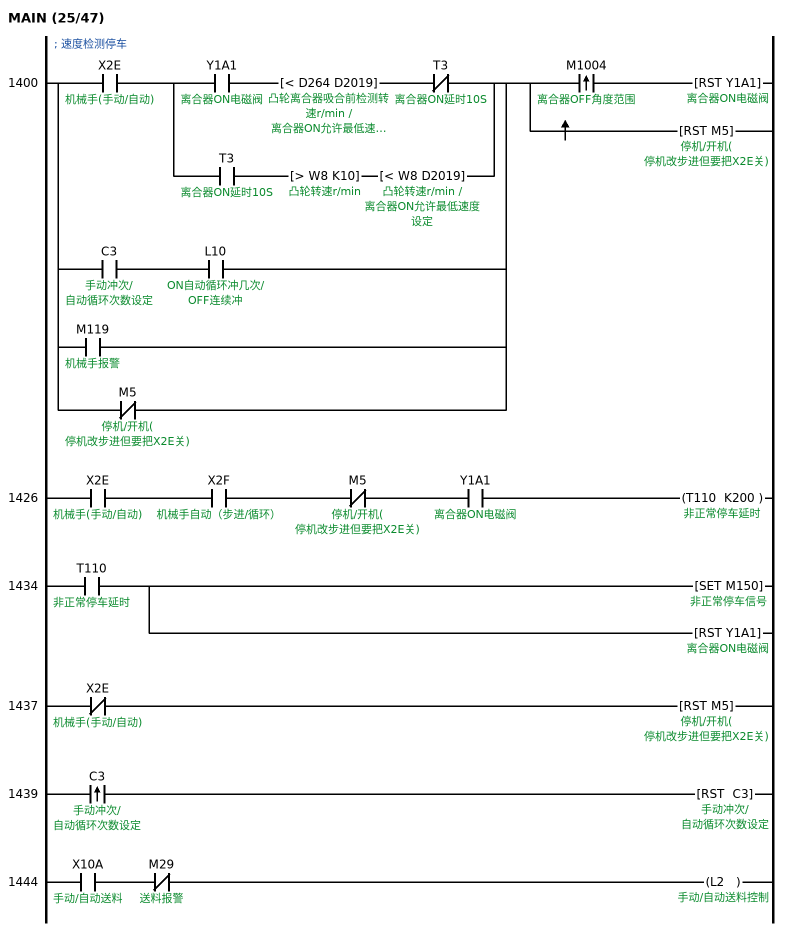
[picture p24: ladder of MAIN, rungs at steps 1400 to 1444]
; 速度检测停车
1400  LD      X2E  ; 机械手(手动/自动)
      LD      Y1A1  ; 离合器ON电磁阀
      AND<    D264 D2019  ; 凸轮离合器吸合前检测转速r/min / 离合器ON允许最低速度设定
      ANI     T3  ; 离合器ON延时10S
      LD      T3  ; 离合器ON延时10S
      AND>    W8 K10  ; 凸轮转速r/min
      AND<    W8 D2019  ; 凸轮转速r/min / 离合器ON允许最低速度设定
      ORB
      ANB
      LD      C3  ; 手动冲次/自动循环次数设定
      AND     L10  ; ON自动循环冲几次/OFF连续冲
      ORB
      OR      M119  ; 机械手报警
      ORI     M5  ; 停机/开机(停机改步进但要把X2E关)
      MPS
      ANDP    M1004  ; 离合器OFF角度范围
      RST     Y1A1  ; 离合器ON电磁阀
      MPP
      MEP
      RST     M5  ; 停机/开机(停机改步进但要把X2E关)
1426  LD      X2E  ; 机械手(手动/自动)
      AND     X2F  ; 机械手自动（步进/循环）
      ANI     M5  ; 停机/开机(停机改步进但要把X2E关)
      AND     Y1A1  ; 离合器ON电磁阀
      OUT     T110 K200  ; 非正常停车延时
1434  LD      T110  ; 非正常停车延时
      SET     M150  ; 非正常停车信号
      RST     Y1A1  ; 离合器ON电磁阀
1437  LDI     X2E  ; 机械手(手动/自动)
      RST     M5  ; 停机/开机(停机改步进但要把X2E关)
1439  LDP     C3  ; 手动冲次/自动循环次数设定
      RST     C3  ; 手动冲次/自动循环次数设定
1444  LD      X10A  ; 手动/自动送料
      ANI     M29  ; 送料报警
      OUT     L2  ; 手动/自动送料控制
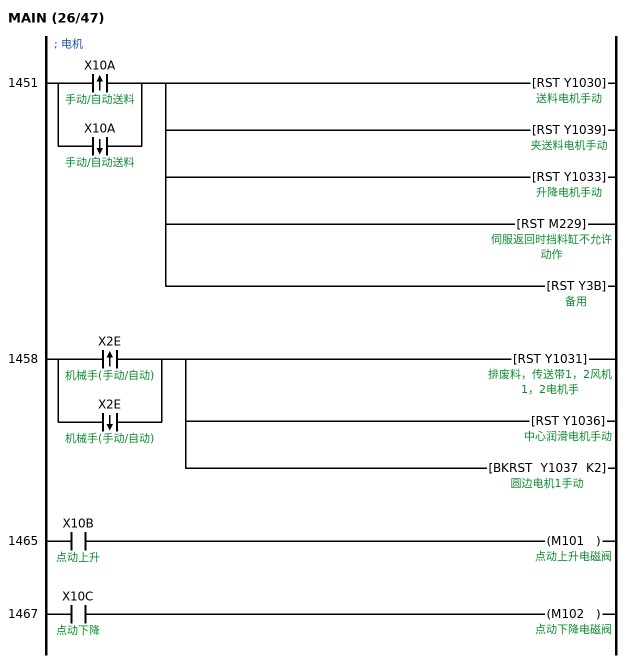
; 电机
1451  LDP     X10A  ; 手动/自动送料
      ORF     X10A  ; 手动/自动送料
      RST     Y1030  ; 送料电机手动
      RST     Y1039  ; 夹送料电机手动
      RST     Y1033  ; 升降电机手动
      RST     M229  ; 伺服返回时挡料缸不允许动作
      RST     Y3B  ; 备用
1458  LDP     X2E  ; 机械手(手动/自动)
      ORF     X2E  ; 机械手(手动/自动)
      RST     Y1031  ; 排废料，传送带1，2风机1，2电机手
      RST     Y1036  ; 中心润滑电机手动
      BKRST   Y1037 K2  ; 圆边电机1手动
1465  LD      X10B  ; 点动上升
      OUT     M101  ; 点动上升电磁阀
1467  LD      X10C  ; 点动下降
      OUT     M102  ; 点动下降电磁阀
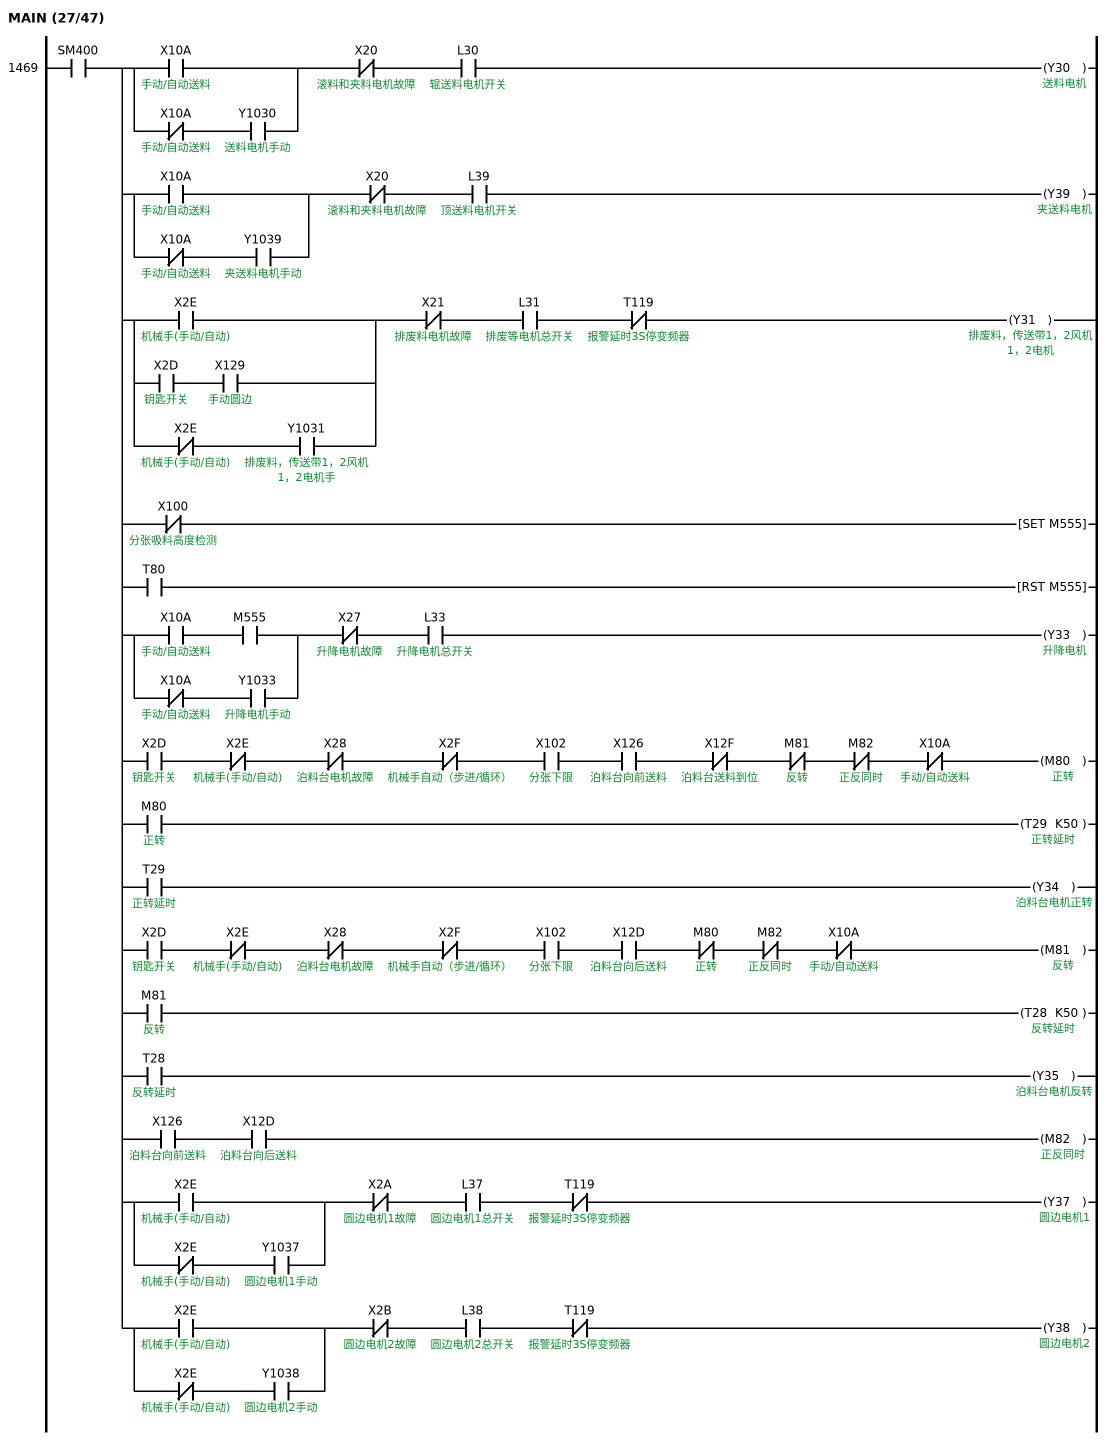
1469  LD      SM400
      MPS
      LD      X10A  ; 手动/自动送料
      LDI     X10A  ; 手动/自动送料
      AND     Y1030  ; 送料电机手动
      ORB
      ANB
      ANI     X20  ; 滚料和夹料电机故障
      AND     L30  ; 辊送料电机开关
      OUT     Y30  ; 送料电机
      MRD
      LD      X10A  ; 手动/自动送料
      LDI     X10A  ; 手动/自动送料
      AND     Y1039  ; 夹送料电机手动
      ORB
      ANB
      ANI     X20  ; 滚料和夹料电机故障
      AND     L39  ; 顶送料电机开关
      OUT     Y39  ; 夹送料电机
      MRD
      LD      X2E  ; 机械手(手动/自动)
      LD      X2D  ; 钥匙开关
      AND     X129  ; 手动圆边
      ORB
      LDI     X2E  ; 机械手(手动/自动)
      AND     Y1031  ; 排废料，传送带1，2风机1，2电机手
      ORB
      ANB
      ANI     X21  ; 排废料电机故障
      AND     L31  ; 排废等电机总开关
      ANI     T119  ; 报警延时3S停变频器
      OUT     Y31  ; 排废料，传送带1，2风机1，2电机
      MRD
      ANI     X100  ; 分张吸料高度检测
      SET     M555
      MRD
      AND     T80
      RST     M555
      MRD
      LD      X10A  ; 手动/自动送料
      AND     M555
      LDI     X10A  ; 手动/自动送料
      AND     Y1033  ; 升降电机手动
      ORB
      ANB
      ANI     X27  ; 升降电机故障
      AND     L33  ; 升降电机总开关
      OUT     Y33  ; 升降电机
      MRD
      AND     X2D  ; 钥匙开关
      ANI     X2E  ; 机械手(手动/自动)
      ANI     X28  ; 泊料台电机故障
      ANI     X2F  ; 机械手自动（步进/循环）
      AND     X102  ; 分张下限
      AND     X126  ; 泊料台向前送料
      ANI     X12F  ; 泊料台送料到位
      ANI     M81  ; 反转
      ANI     M82  ; 正反同时
      ANI     X10A  ; 手动/自动送料
      OUT     M80  ; 正转
      MRD
      AND     M80  ; 正转
      OUT     T29 K50  ; 正转延时
      MRD
      AND     T29  ; 正转延时
      OUT     Y34  ; 泊料台电机正转
      MRD
      AND     X2D  ; 钥匙开关
      ANI     X2E  ; 机械手(手动/自动)
      ANI     X28  ; 泊料台电机故障
      ANI     X2F  ; 机械手自动（步进/循环）
      AND     X102  ; 分张下限
      AND     X12D  ; 泊料台向后送料
      ANI     M80  ; 正转
      ANI     M82  ; 正反同时
      ANI     X10A  ; 手动/自动送料
      OUT     M81  ; 反转
      MRD
      AND     M81  ; 反转
      OUT     T28 K50  ; 反转延时
      MRD
      AND     T28  ; 反转延时
      OUT     Y35  ; 泊料台电机反转
      MRD
      AND     X126  ; 泊料台向前送料
      AND     X12D  ; 泊料台向后送料
      OUT     M82  ; 正反同时
      MRD
      LD      X2E  ; 机械手(手动/自动)
      LDI     X2E  ; 机械手(手动/自动)
      AND     Y1037  ; 圆边电机1手动
      ORB
      ANB
      ANI     X2A  ; 圆边电机1故障
      AND     L37  ; 圆边电机1总开关
      ANI     T119  ; 报警延时3S停变频器
      OUT     Y37  ; 圆边电机1
      MPP
      LD      X2E  ; 机械手(手动/自动)
      LDI     X2E  ; 机械手(手动/自动)
      AND     Y1038  ; 圆边电机2手动
      ORB
      ANB
      ANI     X2B  ; 圆边电机2故障
      AND     L38  ; 圆边电机2总开关
      ANI     T119  ; 报警延时3S停变频器
      OUT     Y38  ; 圆边电机2
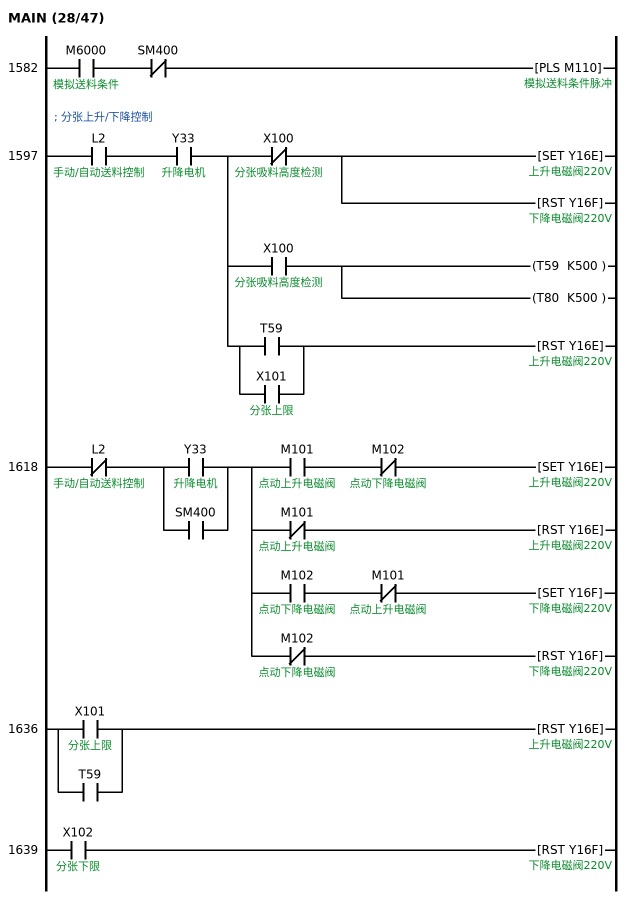
1582  LD      M6000  ; 模拟送料条件
      ANI     SM400
      PLS     M110  ; 模拟送料条件脉冲
; 分张上升/下降控制
1597  LD      L2  ; 手动/自动送料控制
      AND     Y33  ; 升降电机
      MPS
      ANI     X100  ; 分张吸料高度检测
      SET     Y16E  ; 上升电磁阀220V
      RST     Y16F  ; 下降电磁阀220V
      MRD
      AND     X100  ; 分张吸料高度检测
      OUTH    T59 K500
      OUT     T80 K500
      MPP
      LD      T59
      OR      X101  ; 分张上限
      ANB
      RST     Y16E  ; 上升电磁阀220V
1618  LDI     L2  ; 手动/自动送料控制
      LD      Y33  ; 升降电机
      OR      SM400
      ANB
      MPS
      AND     M101  ; 点动上升电磁阀
      ANI     M102  ; 点动下降电磁阀
      SET     Y16E  ; 上升电磁阀220V
      MRD
      ANI     M101  ; 点动上升电磁阀
      RST     Y16E  ; 上升电磁阀220V
      MRD
      AND     M102  ; 点动下降电磁阀
      ANI     M101  ; 点动上升电磁阀
      SET     Y16F  ; 下降电磁阀220V
      MPP
      ANI     M102  ; 点动下降电磁阀
      RST     Y16F  ; 下降电磁阀220V
1636  LD      X101  ; 分张上限
      OR      T59
      RST     Y16E  ; 上升电磁阀220V
1639  LD      X102  ; 分张下限
      RST     Y16F  ; 下降电磁阀220V
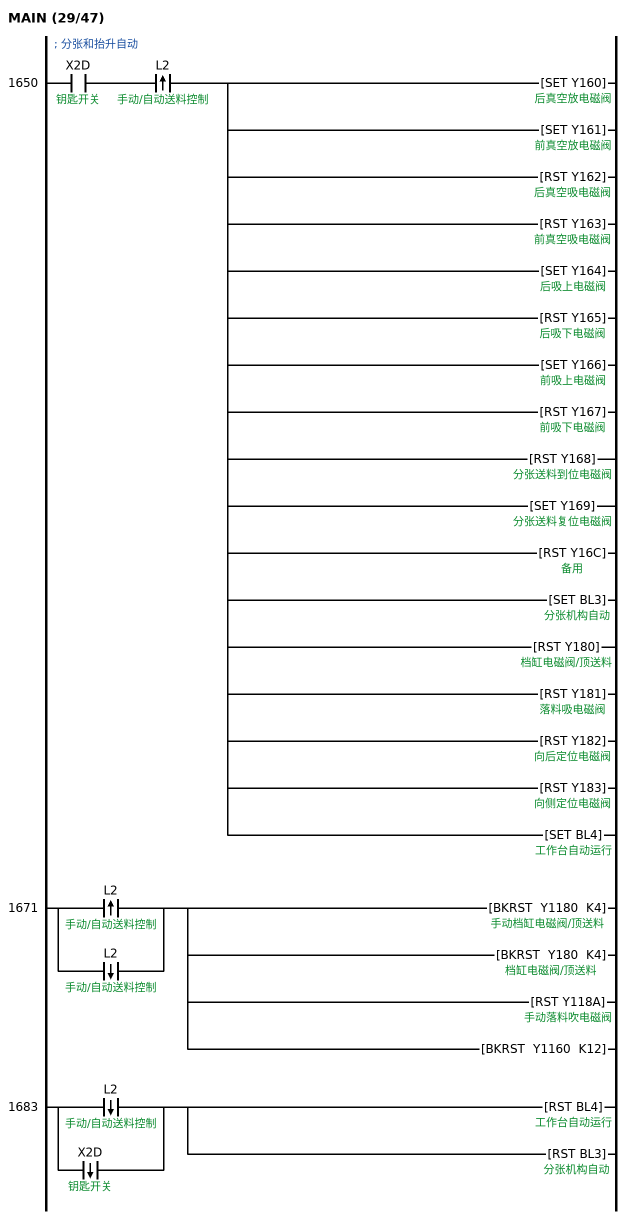
; 分张和抬升自动
1650  LD      X2D  ; 钥匙开关
      ANDP    L2  ; 手动/自动送料控制
      SET     Y160  ; 后真空放电磁阀
      SET     Y161  ; 前真空放电磁阀
      RST     Y162  ; 后真空吸电磁阀
      RST     Y163  ; 前真空吸电磁阀
      SET     Y164  ; 后吸上电磁阀
      RST     Y165  ; 后吸下电磁阀
      SET     Y166  ; 前吸上电磁阀
      RST     Y167  ; 前吸下电磁阀
      RST     Y168  ; 分张送料到位电磁阀
      SET     Y169  ; 分张送料复位电磁阀
      RST     Y16C  ; 备用
      SET     BL3  ; 分张机构自动
      RST     Y180  ; 档缸电磁阀/顶送料
      RST     Y181  ; 落料吸电磁阀
      RST     Y182  ; 向后定位电磁阀
      RST     Y183  ; 向侧定位电磁阀
      SET     BL4  ; 工作台自动运行
1671  LDP     L2  ; 手动/自动送料控制
      ORF     L2  ; 手动/自动送料控制
      BKRST   Y1180 K4  ; 手动档缸电磁阀/顶送料
      BKRST   Y180 K4
      RST     Y118A  ; 手动落料吹电磁阀
      BKRST   Y1160 K12
1683  LDF     L2  ; 手动/自动送料控制
      ORF     X2D  ; 钥匙开关
      RST     BL4  ; 工作台自动运行
      RST     BL3  ; 分张机构自动
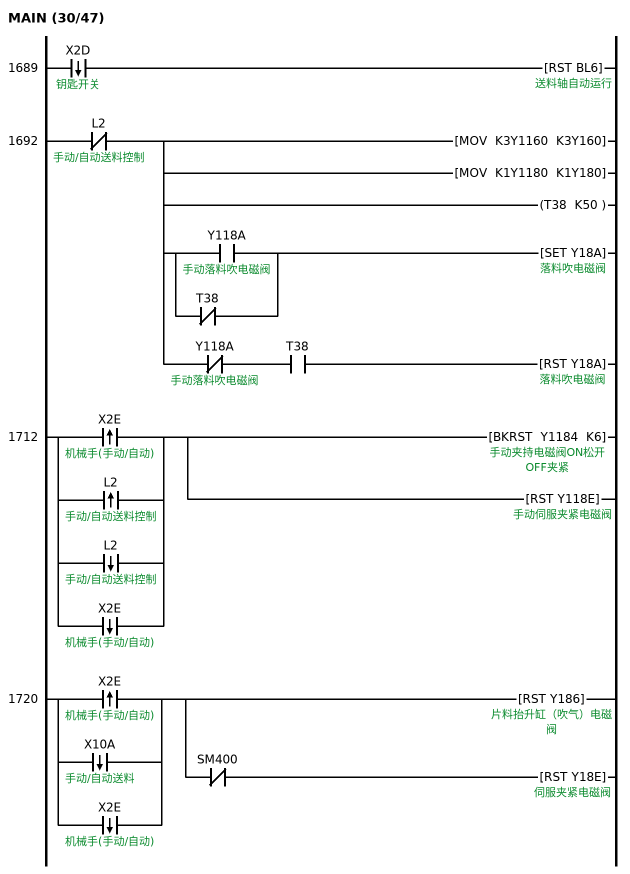
1689  LDF     X2D  ; 钥匙开关
      RST     BL6  ; 送料轴自动运行
1692  LDI     L2  ; 手动/自动送料控制
      MOV     K3Y1160 K3Y160
      MOV     K1Y1180 K1Y180
      OUT     T38 K50
      MPS
      LD      Y118A  ; 手动落料吹电磁阀
      ORI     T38
      ANB
      SET     Y18A  ; 落料吹电磁阀
      MPP
      ANI     Y118A  ; 手动落料吹电磁阀
      AND     T38
      RST     Y18A  ; 落料吹电磁阀
1712  LDP     X2E  ; 机械手(手动/自动)
      ORP     L2  ; 手动/自动送料控制
      ORF     L2  ; 手动/自动送料控制
      ORF     X2E  ; 机械手(手动/自动)
      BKRST   Y1184 K6  ; 手动夹持电磁阀ON松开OFF夹紧
      RST     Y118E  ; 手动伺服夹紧电磁阀
1720  LDP     X2E  ; 机械手(手动/自动)
      ORF     X10A  ; 手动/自动送料
      ORF     X2E  ; 机械手(手动/自动)
      RST     Y186  ; 片料抬升缸（吹气）电磁阀
      ANI     SM400
      RST     Y18E  ; 伺服夹紧电磁阀
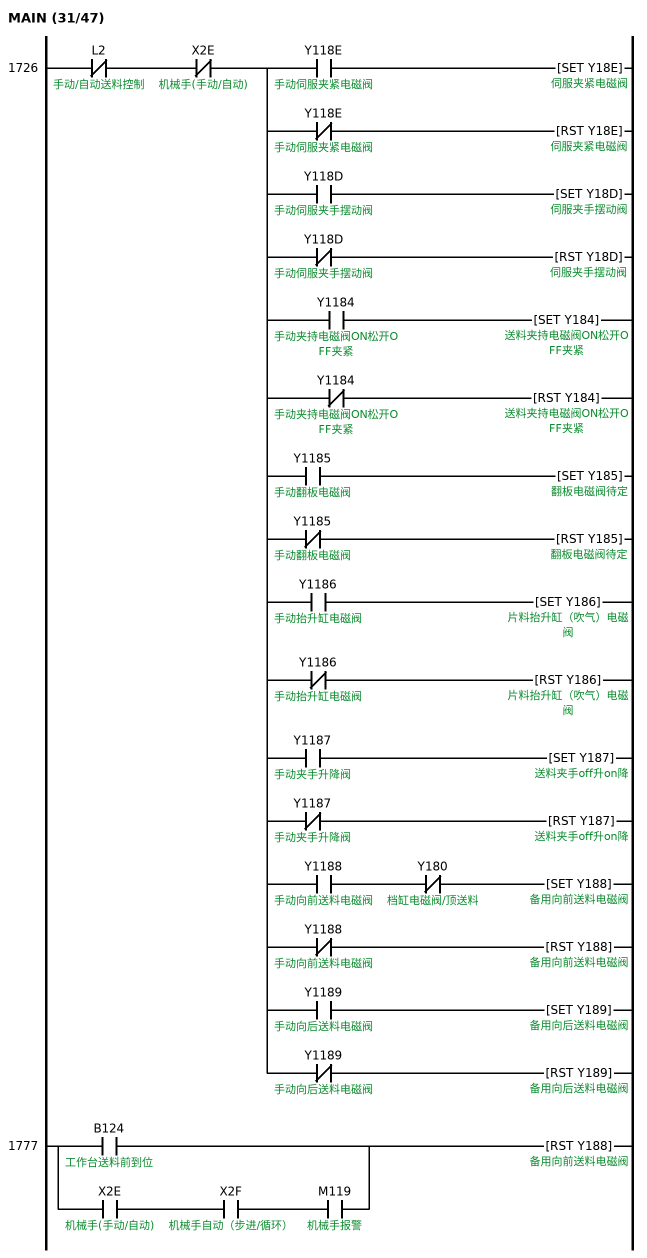
1726  LDI     L2  ; 手动/自动送料控制
      ANI     X2E  ; 机械手(手动/自动)
      MPS
      AND     Y118E  ; 手动伺服夹紧电磁阀
      SET     Y18E  ; 伺服夹紧电磁阀
      MRD
      ANI     Y118E  ; 手动伺服夹紧电磁阀
      RST     Y18E  ; 伺服夹紧电磁阀
      MRD
      AND     Y118D  ; 手动伺服夹手摆动阀
      SET     Y18D  ; 伺服夹手摆动阀
      MRD
      ANI     Y118D  ; 手动伺服夹手摆动阀
      RST     Y18D  ; 伺服夹手摆动阀
      MRD
      AND     Y1184  ; 手动夹持电磁阀ON松开OFF夹紧
      SET     Y184  ; 送料夹持电磁阀ON松开OFF夹紧
      MRD
      ANI     Y1184  ; 手动夹持电磁阀ON松开OFF夹紧
      RST     Y184  ; 送料夹持电磁阀ON松开OFF夹紧
      MRD
      AND     Y1185  ; 手动翻板电磁阀
      SET     Y185  ; 翻板电磁阀待定
      MRD
      ANI     Y1185  ; 手动翻板电磁阀
      RST     Y185  ; 翻板电磁阀待定
      MRD
      AND     Y1186  ; 手动抬升缸电磁阀
      SET     Y186  ; 片料抬升缸（吹气）电磁阀
      MRD
      ANI     Y1186  ; 手动抬升缸电磁阀
      RST     Y186  ; 片料抬升缸（吹气）电磁阀
      MRD
      AND     Y1187  ; 手动夹手升降阀
      SET     Y187  ; 送料夹手off升on降
      MRD
      ANI     Y1187  ; 手动夹手升降阀
      RST     Y187  ; 送料夹手off升on降
      MRD
      AND     Y1188  ; 手动向前送料电磁阀
      ANI     Y180  ; 档缸电磁阀/顶送料
      SET     Y188  ; 备用向前送料电磁阀
      MRD
      ANI     Y1188  ; 手动向前送料电磁阀
      RST     Y188  ; 备用向前送料电磁阀
      MRD
      AND     Y1189  ; 手动向后送料电磁阀
      SET     Y189  ; 备用向后送料电磁阀
      MPP
      ANI     Y1189  ; 手动向后送料电磁阀
      RST     Y189  ; 备用向后送料电磁阀
1777  LD      B124  ; 工作台送料前到位
      LD      X2E  ; 机械手(手动/自动)
      AND     X2F  ; 机械手自动（步进/循环）
      AND     M119  ; 机械手报警
      ORB
      RST     Y188  ; 备用向前送料电磁阀
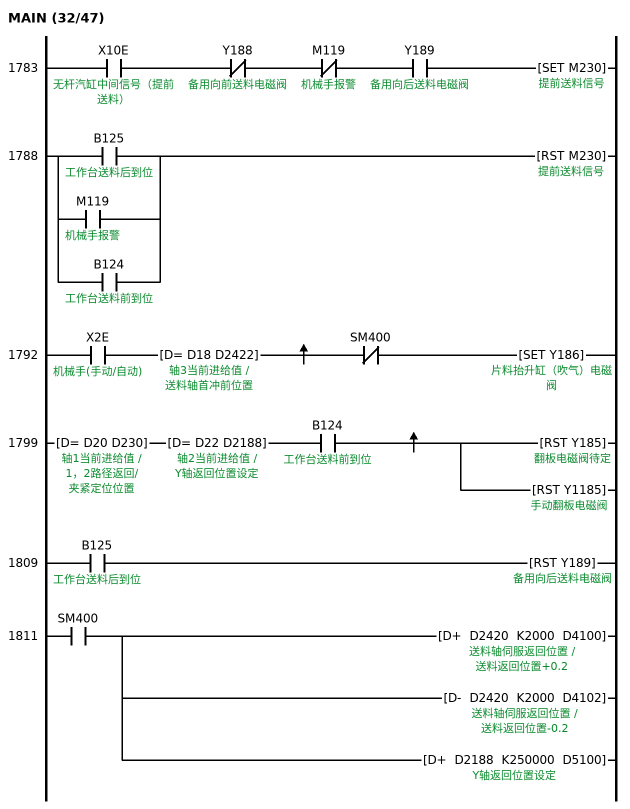
1783  LD      X10E  ; 无杆汽缸中间信号（提前送料）
      ANI     Y188  ; 备用向前送料电磁阀
      ANI     M119  ; 机械手报警
      AND     Y189  ; 备用向后送料电磁阀
      SET     M230  ; 提前送料信号
1788  LD      B125  ; 工作台送料后到位
      OR      M119  ; 机械手报警
      OR      B124  ; 工作台送料前到位
      RST     M230  ; 提前送料信号
1792  LD      X2E  ; 机械手(手动/自动)
      ANDD=   D18 D2422  ; 轴3当前进给值 / 送料轴首冲前位置
      MEP
      ANI     SM400
      SET     Y186  ; 片料抬升缸（吹气）电磁阀
1799  LDD=    D20 D230  ; 轴1当前进给值 / 1，2路径返回/夹紧定位位置
      ANDD=   D22 D2188  ; 轴2当前进给值 / Y轴返回位置设定
      AND     B124  ; 工作台送料前到位
      MEP
      RST     Y185  ; 翻板电磁阀待定
      RST     Y1185  ; 手动翻板电磁阀
1809  LD      B125  ; 工作台送料后到位
      RST     Y189  ; 备用向后送料电磁阀
1811  LD      SM400
      D+      D2420 K2000 D4100  ; 送料返回位置+0.2
      D-      D2420 K2000 D4102  ; 送料返回位置-0.2
      D+      D2188 K250000 D5100
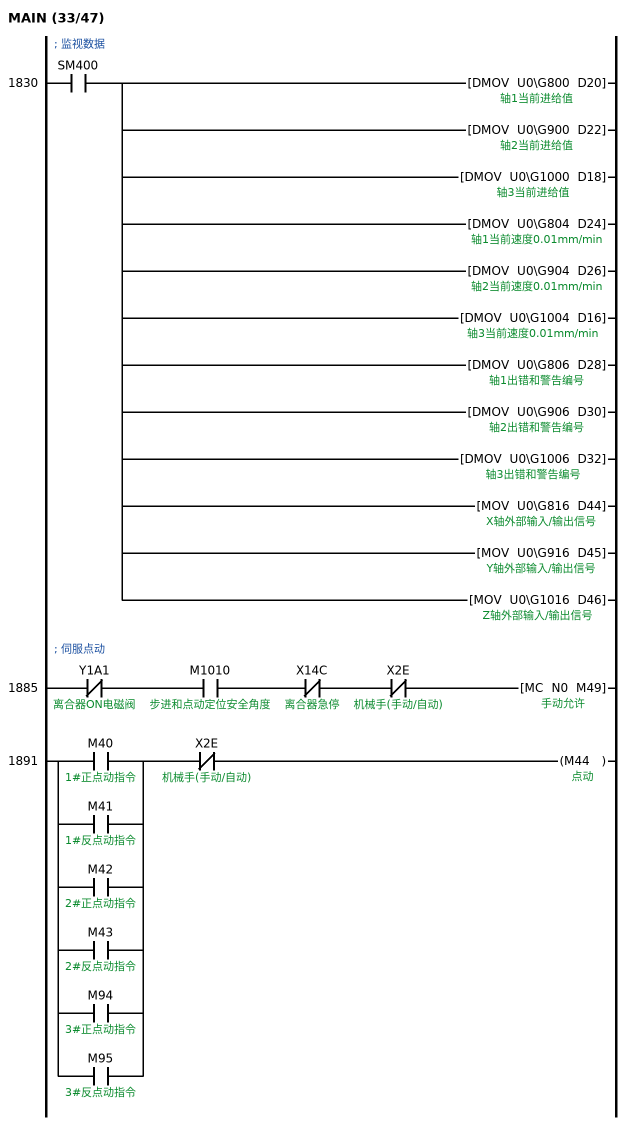
; 监视数据
1830  LD      SM400
      DMOV    U0\G800 D20
      DMOV    U0\G900 D22
      DMOV    U0\G1000 D18
      DMOV    U0\G804 D24  ; 轴1当前速度0.01mm/min
      DMOV    U0\G904 D26  ; 轴2当前速度0.01mm/min
      DMOV    U0\G1004 D16  ; 轴3当前速度0.01mm/min
      DMOV    U0\G806 D28
      DMOV    U0\G906 D30
      DMOV    U0\G1006 D32  ; 轴3出错和警告编号
      MOV     U0\G816 D44  ; X轴外部输入/输出信号
      MOV     U0\G916 D45  ; Y轴外部输入/输出信号
      MOV     U0\G1016 D46  ; Z轴外部输入/输出信号
; 伺服点动
1885  LDI     Y1A1  ; 离合器ON电磁阀
      AND     M1010  ; 步进和点动定位安全角度
      ANI     X14C  ; 离合器急停
      ANI     X2E  ; 机械手(手动/自动)
      MC      N0 M49  ; 手动允许
1891  LD      M40  ; 1#正点动指令
      OR      M41  ; 1#反点动指令
      OR      M42  ; 2#正点动指令
      OR      M43  ; 2#反点动指令
      OR      M94  ; 3#正点动指令
      OR      M95  ; 3#反点动指令
      ANI     X2E  ; 机械手(手动/自动)
      OUT     M44  ; 点动
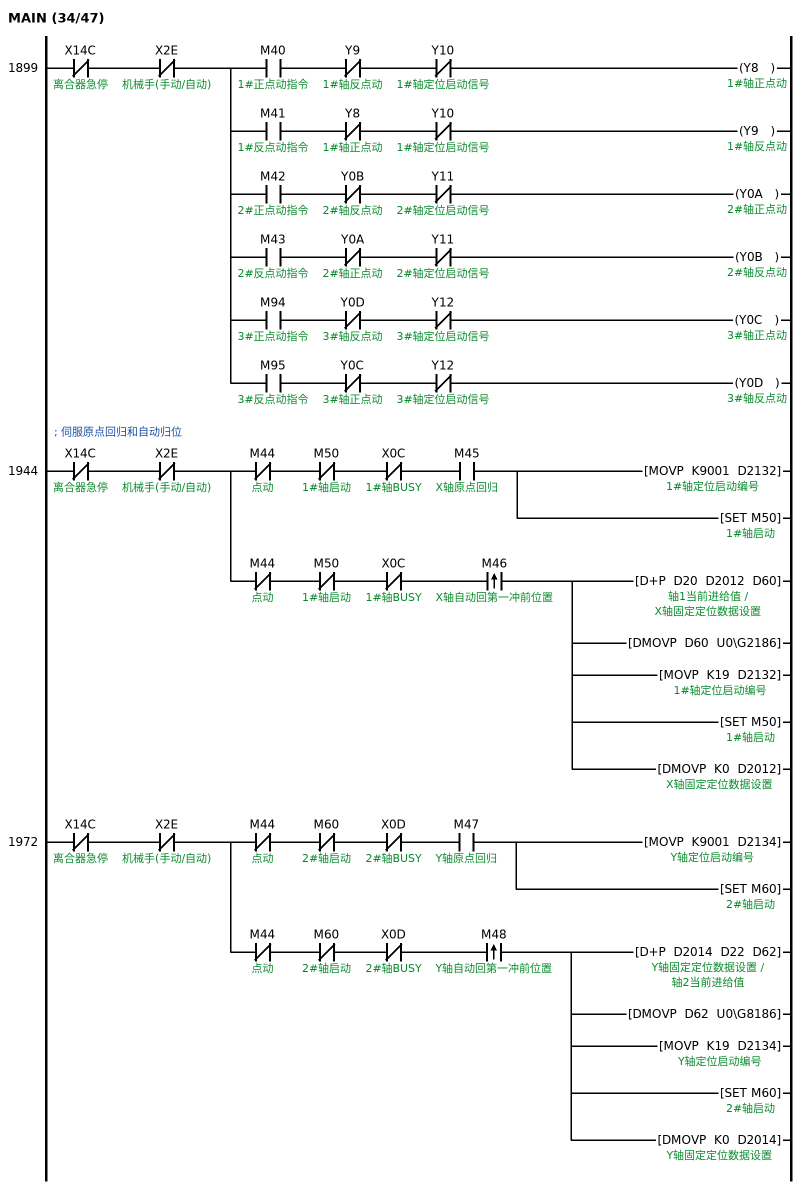
1899  LDI     X14C  ; 离合器急停
      ANI     X2E  ; 机械手(手动/自动)
      MPS
      AND     M40  ; 1#正点动指令
      ANI     Y9  ; 1#轴反点动
      ANI     Y10  ; 1#轴定位启动信号
      OUT     Y8  ; 1#轴正点动
      MRD
      AND     M41  ; 1#反点动指令
      ANI     Y8  ; 1#轴正点动
      ANI     Y10  ; 1#轴定位启动信号
      OUT     Y9  ; 1#轴反点动
      MRD
      AND     M42  ; 2#正点动指令
      ANI     Y0B  ; 2#轴反点动
      ANI     Y11  ; 2#轴定位启动信号
      OUT     Y0A  ; 2#轴正点动
      MRD
      AND     M43  ; 2#反点动指令
      ANI     Y0A  ; 2#轴正点动
      ANI     Y11  ; 2#轴定位启动信号
      OUT     Y0B  ; 2#轴反点动
      MRD
      AND     M94  ; 3#正点动指令
      ANI     Y0D  ; 3#轴反点动
      ANI     Y12  ; 3#轴定位启动信号
      OUT     Y0C  ; 3#轴正点动
      MPP
      AND     M95  ; 3#反点动指令
      ANI     Y0C  ; 3#轴正点动
      ANI     Y12  ; 3#轴定位启动信号
      OUT     Y0D  ; 3#轴反点动
; 伺服原点回归和自动归位
1944  LDI     X14C  ; 离合器急停
      ANI     X2E  ; 机械手(手动/自动)
      MPS
      ANI     M44  ; 点动
      ANI     M50  ; 1#轴启动
      ANI     X0C  ; 1#轴BUSY
      AND     M45  ; X轴原点回归
      MOVP    K9001 D2132  ; 1#轴定位启动编号
      SET     M50  ; 1#轴启动
      MPP
      ANI     M44  ; 点动
      ANI     M50  ; 1#轴启动
      ANI     X0C  ; 1#轴BUSY
      ANDP    M46  ; X轴自动回第一冲前位置
      D+P     D20 D2012 D60  ; X轴固定定位数据设置
      DMOVP   D60 U0\G2186
      MOVP    K19 D2132
      SET     M50  ; 1#轴启动
      DMOVP   K0 D2012
1972  LDI     X14C  ; 离合器急停
      ANI     X2E  ; 机械手(手动/自动)
      MPS
      ANI     M44  ; 点动
      ANI     M60  ; 2#轴启动
      ANI     X0D  ; 2#轴BUSY
      AND     M47  ; Y轴原点回归
      MOVP    K9001 D2134  ; Y轴定位启动编号
      SET     M60  ; 2#轴启动
      MPP
      ANI     M44  ; 点动
      ANI     M60  ; 2#轴启动
      ANI     X0D  ; 2#轴BUSY
      ANDP    M48  ; Y轴自动回第一冲前位置
      D+P     D2014 D22 D62  ; Y轴固定定位数据设置
      DMOVP   D62 U0\G8186
      MOVP    K19 D2134
      SET     M60  ; 2#轴启动
      DMOVP   K0 D2014
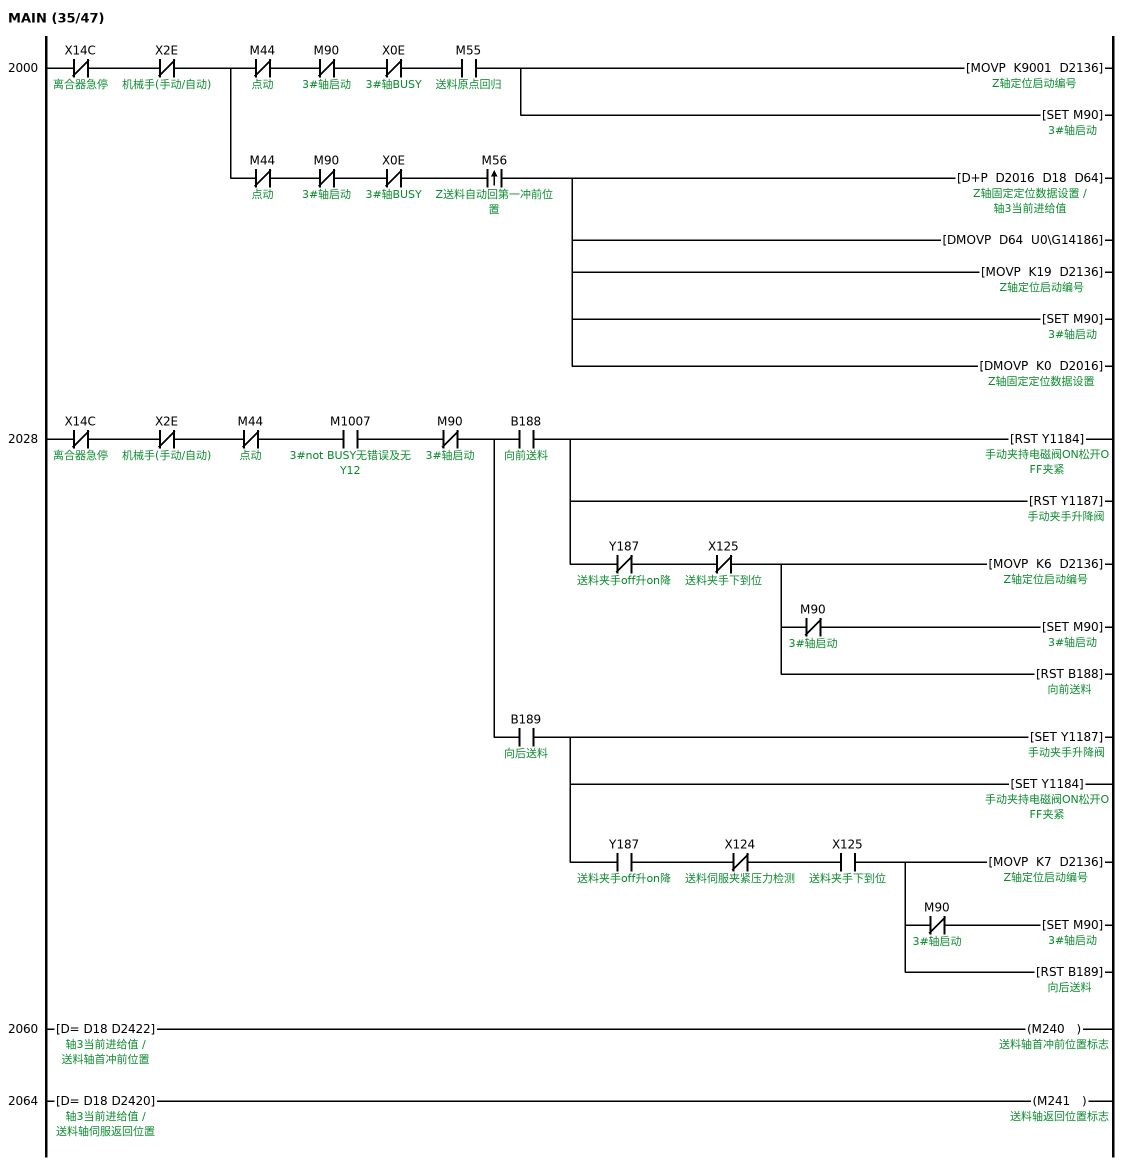
2000  LDI     X14C  ; 离合器急停
      ANI     X2E  ; 机械手(手动/自动)
      MPS
      ANI     M44  ; 点动
      ANI     M90  ; 3#轴启动
      ANI     X0E  ; 3#轴BUSY
      AND     M55  ; 送料原点回归
      MOVP    K9001 D2136  ; Z轴定位启动编号
      SET     M90  ; 3#轴启动
      MPP
      ANI     M44  ; 点动
      ANI     M90  ; 3#轴启动
      ANI     X0E  ; 3#轴BUSY
      ANDP    M56  ; Z送料自动回第一冲前位置
      D+P     D2016 D18 D64  ; Z轴固定定位数据设置
      DMOVP   D64 U0\G14186
      MOVP    K19 D2136
      SET     M90  ; 3#轴启动
      DMOVP   K0 D2016
2028  LDI     X14C  ; 离合器急停
      ANI     X2E  ; 机械手(手动/自动)
      ANI     M44  ; 点动
      AND     M1007  ; 3#not BUSY无错误及无Y12
      ANI     M90  ; 3#轴启动
      MPS
      AND     B188  ; 向前送料
      RST     Y1184  ; 手动夹持电磁阀ON松开OFF夹紧
      RST     Y1187  ; 手动夹手升降阀
      ANI     Y187  ; 送料夹手off升on降
      ANI     X125  ; 送料夹手下到位
      MOVP    K6 D2136
      MPS
      ANI     M90  ; 3#轴启动
      SET     M90  ; 3#轴启动
      MPP
      RST     B188  ; 向前送料
      MPP
      AND     B189  ; 向后送料
      SET     Y1187  ; 手动夹手升降阀
      SET     Y1184  ; 手动夹持电磁阀ON松开OFF夹紧
      AND     Y187  ; 送料夹手off升on降
      ANI     X124  ; 送料伺服夹紧压力检测
      AND     X125  ; 送料夹手下到位
      MOVP    K7 D2136
      MPS
      ANI     M90  ; 3#轴启动
      SET     M90  ; 3#轴启动
      MPP
      RST     B189  ; 向后送料
2060  LDD=    D18 D2422  ; 轴3当前进给值 / 送料轴首冲前位置
      OUT     M240  ; 送料轴首冲前位置标志
2064  LDD=    D18 D2420  ; 轴3当前进给值 / 送料轴伺服返回位置
      OUT     M241  ; 送料轴返回位置标志
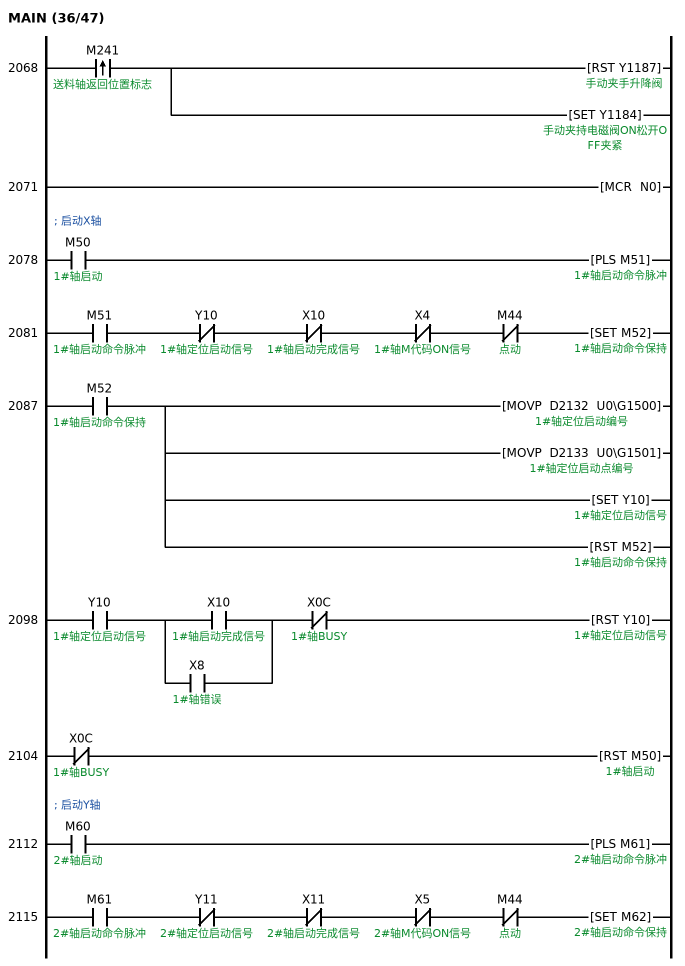
2068  LDP     M241  ; 送料轴返回位置标志
      RST     Y1187  ; 手动夹手升降阀
      SET     Y1184  ; 手动夹持电磁阀ON松开OFF夹紧
2071  MCR     N0
; 启动X轴
2078  LD      M50  ; 1#轴启动
      PLS     M51  ; 1#轴启动命令脉冲
2081  LD      M51  ; 1#轴启动命令脉冲
      ANI     Y10  ; 1#轴定位启动信号
      ANI     X10  ; 1#轴启动完成信号
      ANI     X4  ; 1#轴M代码ON信号
      ANI     M44  ; 点动
      SET     M52  ; 1#轴启动命令保持
2087  LD      M52  ; 1#轴启动命令保持
      MOVP    D2132 U0\G1500
      MOVP    D2133 U0\G1501  ; 1#轴定位启动点编号
      SET     Y10  ; 1#轴定位启动信号
      RST     M52  ; 1#轴启动命令保持
2098  LD      Y10  ; 1#轴定位启动信号
      LD      X10  ; 1#轴启动完成信号
      OR      X8  ; 1#轴错误
      ANB
      ANI     X0C  ; 1#轴BUSY
      RST     Y10  ; 1#轴定位启动信号
2104  LDI     X0C  ; 1#轴BUSY
      RST     M50  ; 1#轴启动
; 启动Y轴
2112  LD      M60  ; 2#轴启动
      PLS     M61  ; 2#轴启动命令脉冲
2115  LD      M61  ; 2#轴启动命令脉冲
      ANI     Y11  ; 2#轴定位启动信号
      ANI     X11  ; 2#轴启动完成信号
      ANI     X5  ; 2#轴M代码ON信号
      ANI     M44  ; 点动
      SET     M62  ; 2#轴启动命令保持
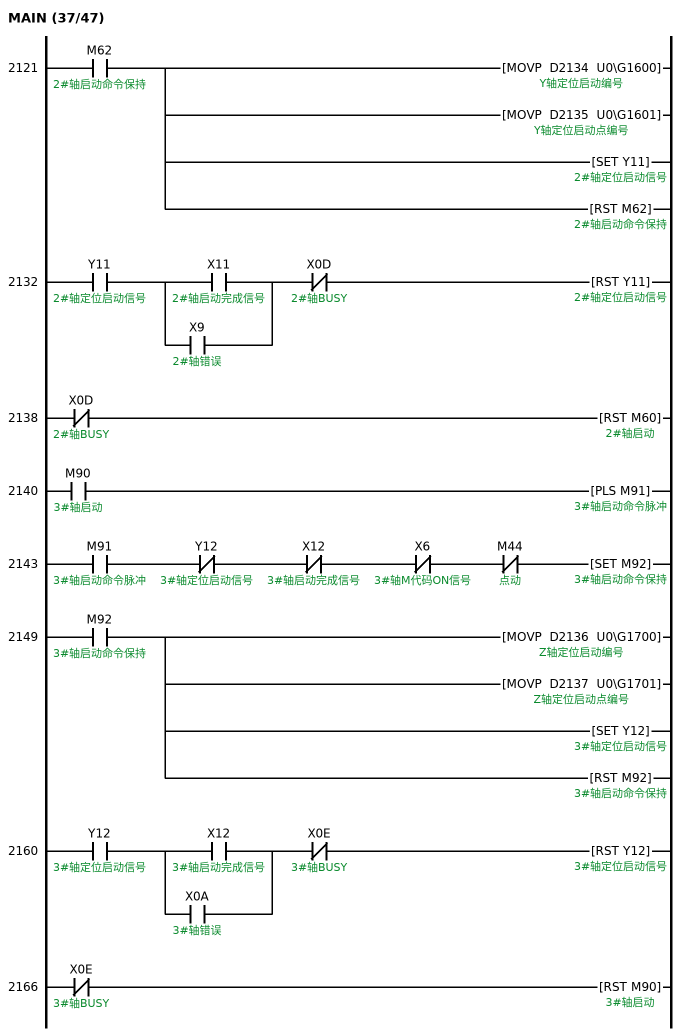
2121  LD      M62  ; 2#轴启动命令保持
      MOVP    D2134 U0\G1600
      MOVP    D2135 U0\G1601  ; Y轴定位启动点编号
      SET     Y11  ; 2#轴定位启动信号
      RST     M62  ; 2#轴启动命令保持
2132  LD      Y11  ; 2#轴定位启动信号
      LD      X11  ; 2#轴启动完成信号
      OR      X9  ; 2#轴错误
      ANB
      ANI     X0D  ; 2#轴BUSY
      RST     Y11  ; 2#轴定位启动信号
2138  LDI     X0D  ; 2#轴BUSY
      RST     M60  ; 2#轴启动
2140  LD      M90  ; 3#轴启动
      PLS     M91  ; 3#轴启动命令脉冲
2143  LD      M91  ; 3#轴启动命令脉冲
      ANI     Y12  ; 3#轴定位启动信号
      ANI     X12  ; 3#轴启动完成信号
      ANI     X6  ; 3#轴M代码ON信号
      ANI     M44  ; 点动
      SET     M92  ; 3#轴启动命令保持
2149  LD      M92  ; 3#轴启动命令保持
      MOVP    D2136 U0\G1700
      MOVP    D2137 U0\G1701  ; Z轴定位启动点编号
      SET     Y12  ; 3#轴定位启动信号
      RST     M92  ; 3#轴启动命令保持
2160  LD      Y12  ; 3#轴定位启动信号
      LD      X12  ; 3#轴启动完成信号
      OR      X0A  ; 3#轴错误
      ANB
      ANI     X0E  ; 3#轴BUSY
      RST     Y12  ; 3#轴定位启动信号
2166  LDI     X0E  ; 3#轴BUSY
      RST     M90  ; 3#轴启动
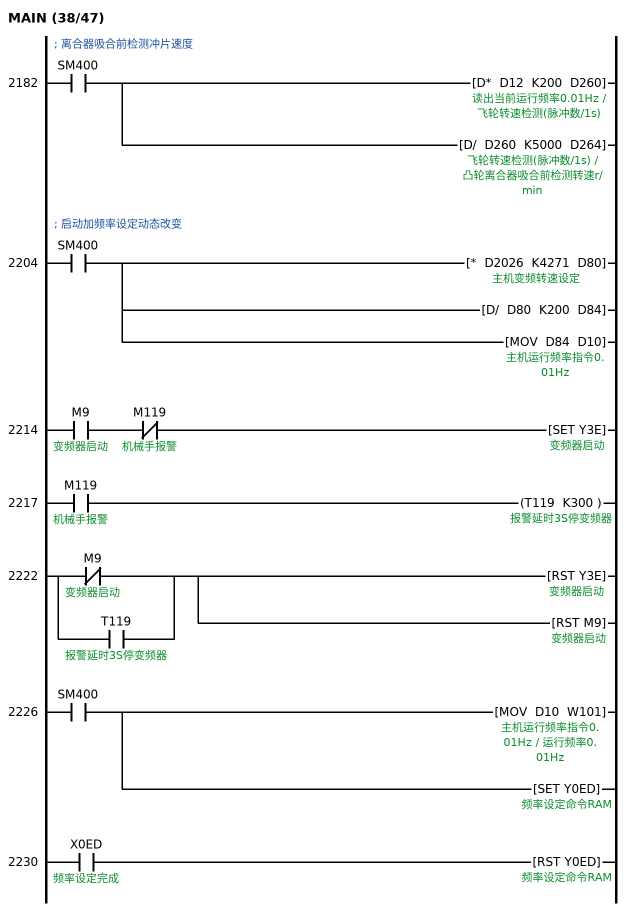
; 离合器吸合前检测冲片速度
2182  LD      SM400
      D*      D12 K200 D260  ; 读出当前运行频率0.01Hz / 飞轮转速检测(脉冲数/1s)
      D/      D260 K5000 D264
; 启动加频率设定动态改变
2204  LD      SM400
      *       D2026 K4271 D80  ; 主机变频转速设定
      D/      D80 K200 D84
      MOV     D84 D10  ; 主机运行频率指令0.01Hz
2214  LD      M9  ; 变频器启动
      ANI     M119  ; 机械手报警
      SET     Y3E  ; 变频器启动
2217  LD      M119  ; 机械手报警
      OUT     T119 K300  ; 报警延时3S停变频器
2222  LDI     M9  ; 变频器启动
      OR      T119  ; 报警延时3S停变频器
      RST     Y3E  ; 变频器启动
      RST     M9  ; 变频器启动
2226  LD      SM400
      MOV     D10 W101  ; 运行频率0.01Hz
      SET     Y0ED  ; 频率设定命令RAM
2230  LD      X0ED  ; 频率设定完成
      RST     Y0ED  ; 频率设定命令RAM
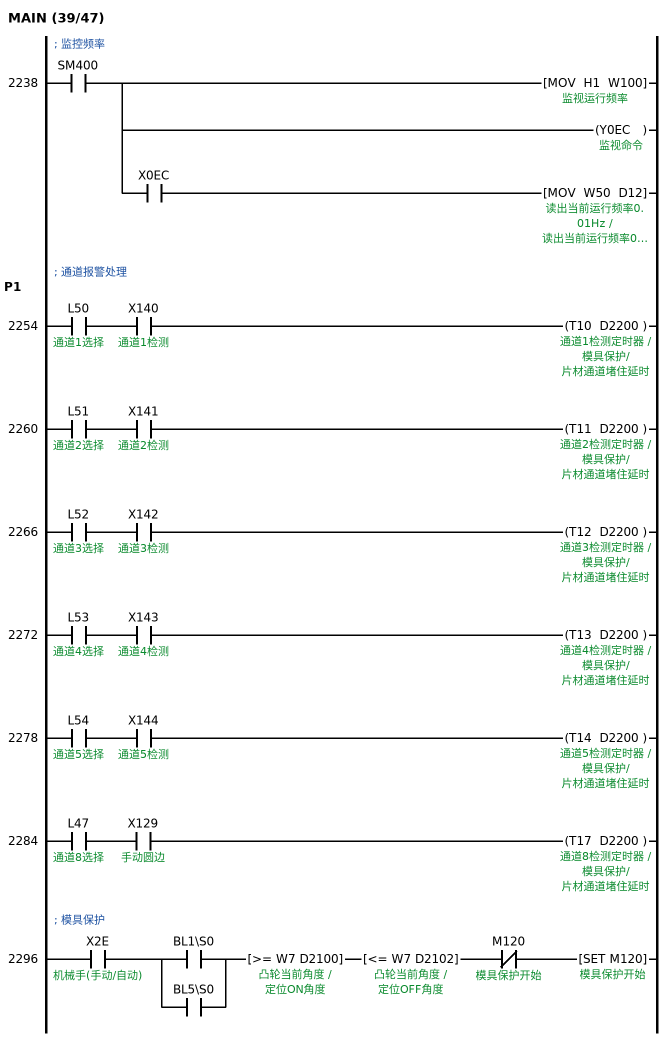
; 监控频率
2238  LD      SM400
      MOV     H1 W100  ; 监视运行频率
      OUT     Y0EC  ; 监视命令
      AND     X0EC
      MOV     W50 D12  ; 读出当前运行频率0.01Hz
; 通道报警处理
      P1
2254  LD      L50  ; 通道1选择
      AND     X140  ; 通道1检测
      OUTH    T10 D2200  ; 通道1检测定时器 / 模具保护/片材通道堵住延时
2260  LD      L51  ; 通道2选择
      AND     X141  ; 通道2检测
      OUTH    T11 D2200  ; 通道2检测定时器 / 模具保护/片材通道堵住延时
2266  LD      L52  ; 通道3选择
      AND     X142  ; 通道3检测
      OUTH    T12 D2200  ; 通道3检测定时器 / 模具保护/片材通道堵住延时
2272  LD      L53  ; 通道4选择
      AND     X143  ; 通道4检测
      OUTH    T13 D2200  ; 通道4检测定时器 / 模具保护/片材通道堵住延时
2278  LD      L54  ; 通道5选择
      AND     X144  ; 通道5检测
      OUTH    T14 D2200  ; 通道5检测定时器 / 模具保护/片材通道堵住延时
2284  LD      L47  ; 通道8选择
      AND     X129  ; 手动圆边
      OUTH    T17 D2200  ; 通道8检测定时器 / 模具保护/片材通道堵住延时
; 模具保护
2296  LD      X2E  ; 机械手(手动/自动)
      LD      BL1\S0
      OR      BL5\S0
      ANB
      AND>=   W7 D2100  ; 凸轮当前角度 / 定位ON角度
      AND<=   W7 D2102  ; 凸轮当前角度 / 定位OFF角度
      ANI     M120  ; 模具保护开始
      SET     M120  ; 模具保护开始
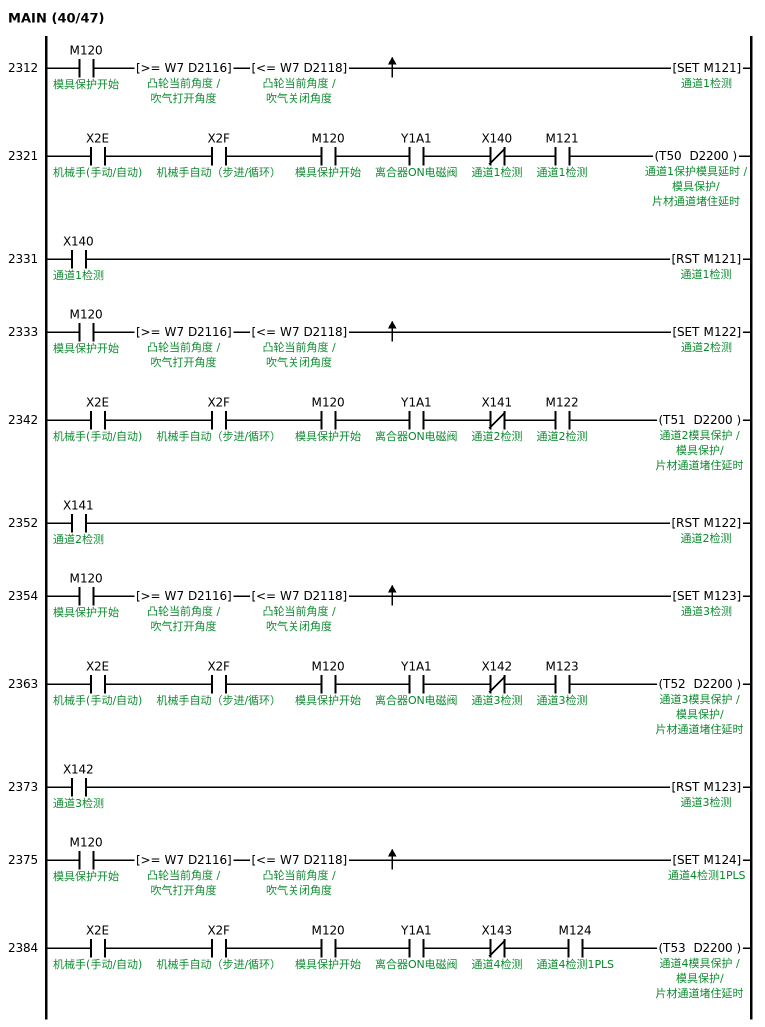
2312  LD      M120  ; 模具保护开始
      AND>=   W7 D2116  ; 凸轮当前角度 / 吹气打开角度
      AND<=   W7 D2118  ; 凸轮当前角度 / 吹气关闭角度
      MEP
      SET     M121  ; 通道1检测
2321  LD      X2E  ; 机械手(手动/自动)
      AND     X2F  ; 机械手自动（步进/循环）
      AND     M120  ; 模具保护开始
      AND     Y1A1  ; 离合器ON电磁阀
      ANI     X140  ; 通道1检测
      AND     M121  ; 通道1检测
      OUTH    T50 D2200  ; 通道1保护模具延时 / 模具保护/片材通道堵住延时
2331  LD      X140  ; 通道1检测
      RST     M121  ; 通道1检测
2333  LD      M120  ; 模具保护开始
      AND>=   W7 D2116  ; 凸轮当前角度 / 吹气打开角度
      AND<=   W7 D2118  ; 凸轮当前角度 / 吹气关闭角度
      MEP
      SET     M122  ; 通道2检测
2342  LD      X2E  ; 机械手(手动/自动)
      AND     X2F  ; 机械手自动（步进/循环）
      AND     M120  ; 模具保护开始
      AND     Y1A1  ; 离合器ON电磁阀
      ANI     X141  ; 通道2检测
      AND     M122  ; 通道2检测
      OUTH    T51 D2200  ; 通道2模具保护 / 模具保护/片材通道堵住延时
2352  LD      X141  ; 通道2检测
      RST     M122  ; 通道2检测
2354  LD      M120  ; 模具保护开始
      AND>=   W7 D2116  ; 凸轮当前角度 / 吹气打开角度
      AND<=   W7 D2118  ; 凸轮当前角度 / 吹气关闭角度
      MEP
      SET     M123  ; 通道3检测
2363  LD      X2E  ; 机械手(手动/自动)
      AND     X2F  ; 机械手自动（步进/循环）
      AND     M120  ; 模具保护开始
      AND     Y1A1  ; 离合器ON电磁阀
      ANI     X142  ; 通道3检测
      AND     M123  ; 通道3检测
      OUTH    T52 D2200  ; 通道3模具保护 / 模具保护/片材通道堵住延时
2373  LD      X142  ; 通道3检测
      RST     M123  ; 通道3检测
2375  LD      M120  ; 模具保护开始
      AND>=   W7 D2116  ; 凸轮当前角度 / 吹气打开角度
      AND<=   W7 D2118  ; 凸轮当前角度 / 吹气关闭角度
      MEP
      SET     M124  ; 通道4检测1PLS
2384  LD      X2E  ; 机械手(手动/自动)
      AND     X2F  ; 机械手自动（步进/循环）
      AND     M120  ; 模具保护开始
      AND     Y1A1  ; 离合器ON电磁阀
      ANI     X143  ; 通道4检测
      AND     M124  ; 通道4检测1PLS
      OUTH    T53 D2200  ; 通道4模具保护 / 模具保护/片材通道堵住延时
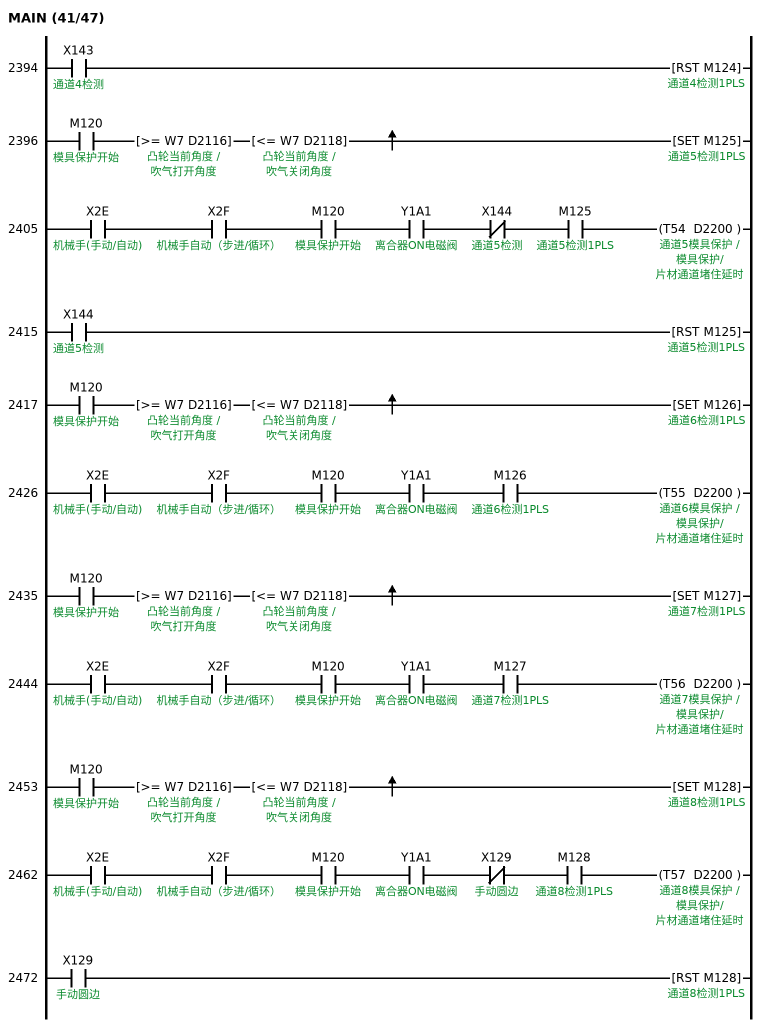
2394  LD      X143  ; 通道4检测
      RST     M124  ; 通道4检测1PLS
2396  LD      M120  ; 模具保护开始
      AND>=   W7 D2116  ; 凸轮当前角度 / 吹气打开角度
      AND<=   W7 D2118  ; 凸轮当前角度 / 吹气关闭角度
      MEP
      SET     M125  ; 通道5检测1PLS
2405  LD      X2E  ; 机械手(手动/自动)
      AND     X2F  ; 机械手自动（步进/循环）
      AND     M120  ; 模具保护开始
      AND     Y1A1  ; 离合器ON电磁阀
      ANI     X144  ; 通道5检测
      AND     M125  ; 通道5检测1PLS
      OUTH    T54 D2200  ; 通道5模具保护 / 模具保护/片材通道堵住延时
2415  LD      X144  ; 通道5检测
      RST     M125  ; 通道5检测1PLS
2417  LD      M120  ; 模具保护开始
      AND>=   W7 D2116  ; 凸轮当前角度 / 吹气打开角度
      AND<=   W7 D2118  ; 凸轮当前角度 / 吹气关闭角度
      MEP
      SET     M126  ; 通道6检测1PLS
2426  LD      X2E  ; 机械手(手动/自动)
      AND     X2F  ; 机械手自动（步进/循环）
      AND     M120  ; 模具保护开始
      AND     Y1A1  ; 离合器ON电磁阀
      AND     M126  ; 通道6检测1PLS
      OUTH    T55 D2200  ; 通道6模具保护 / 模具保护/片材通道堵住延时
2435  LD      M120  ; 模具保护开始
      AND>=   W7 D2116  ; 凸轮当前角度 / 吹气打开角度
      AND<=   W7 D2118  ; 凸轮当前角度 / 吹气关闭角度
      MEP
      SET     M127  ; 通道7检测1PLS
2444  LD      X2E  ; 机械手(手动/自动)
      AND     X2F  ; 机械手自动（步进/循环）
      AND     M120  ; 模具保护开始
      AND     Y1A1  ; 离合器ON电磁阀
      AND     M127  ; 通道7检测1PLS
      OUTH    T56 D2200  ; 通道7模具保护 / 模具保护/片材通道堵住延时
2453  LD      M120  ; 模具保护开始
      AND>=   W7 D2116  ; 凸轮当前角度 / 吹气打开角度
      AND<=   W7 D2118  ; 凸轮当前角度 / 吹气关闭角度
      MEP
      SET     M128  ; 通道8检测1PLS
2462  LD      X2E  ; 机械手(手动/自动)
      AND     X2F  ; 机械手自动（步进/循环）
      AND     M120  ; 模具保护开始
      AND     Y1A1  ; 离合器ON电磁阀
      ANI     X129  ; 手动圆边
      AND     M128  ; 通道8检测1PLS
      OUTH    T57 D2200  ; 通道8模具保护 / 模具保护/片材通道堵住延时
2472  LD      X129  ; 手动圆边
      RST     M128  ; 通道8检测1PLS
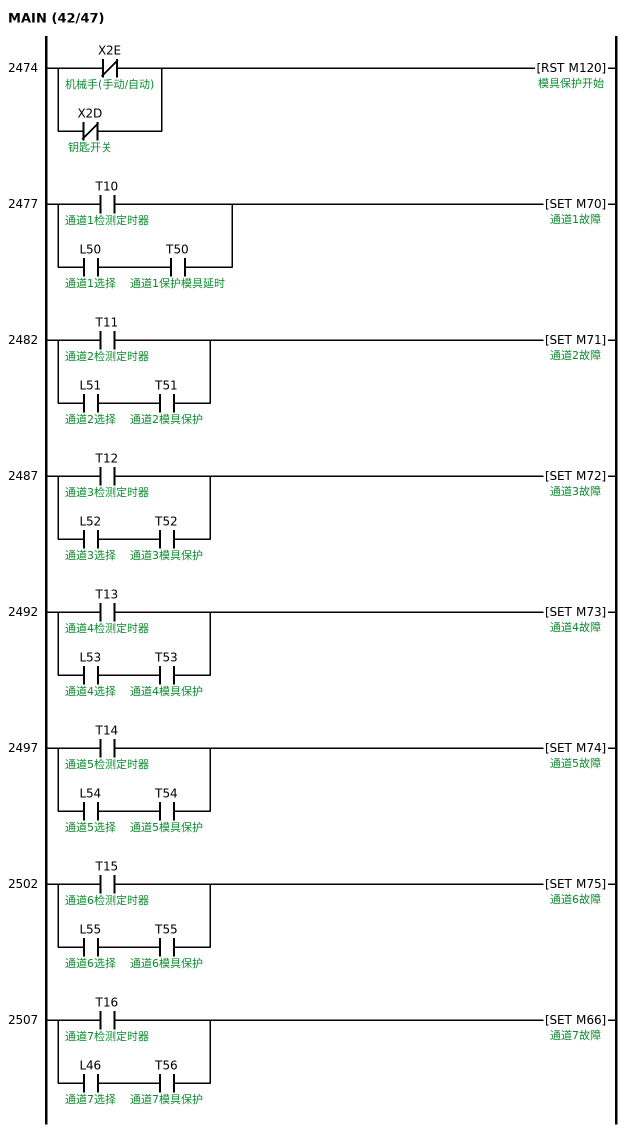
2474  LDI     X2E  ; 机械手(手动/自动)
      ORI     X2D  ; 钥匙开关
      RST     M120  ; 模具保护开始
2477  LD      T10  ; 通道1检测定时器
      LD      L50  ; 通道1选择
      AND     T50  ; 通道1保护模具延时
      ORB
      SET     M70  ; 通道1故障
2482  LD      T11  ; 通道2检测定时器
      LD      L51  ; 通道2选择
      AND     T51  ; 通道2模具保护
      ORB
      SET     M71  ; 通道2故障
2487  LD      T12  ; 通道3检测定时器
      LD      L52  ; 通道3选择
      AND     T52  ; 通道3模具保护
      ORB
      SET     M72  ; 通道3故障
2492  LD      T13  ; 通道4检测定时器
      LD      L53  ; 通道4选择
      AND     T53  ; 通道4模具保护
      ORB
      SET     M73  ; 通道4故障
2497  LD      T14  ; 通道5检测定时器
      LD      L54  ; 通道5选择
      AND     T54  ; 通道5模具保护
      ORB
      SET     M74  ; 通道5故障
2502  LD      T15  ; 通道6检测定时器
      LD      L55  ; 通道6选择
      AND     T55  ; 通道6模具保护
      ORB
      SET     M75  ; 通道6故障
2507  LD      T16  ; 通道7检测定时器
      LD      L46  ; 通道7选择
      AND     T56  ; 通道7模具保护
      ORB
      SET     M66  ; 通道7故障
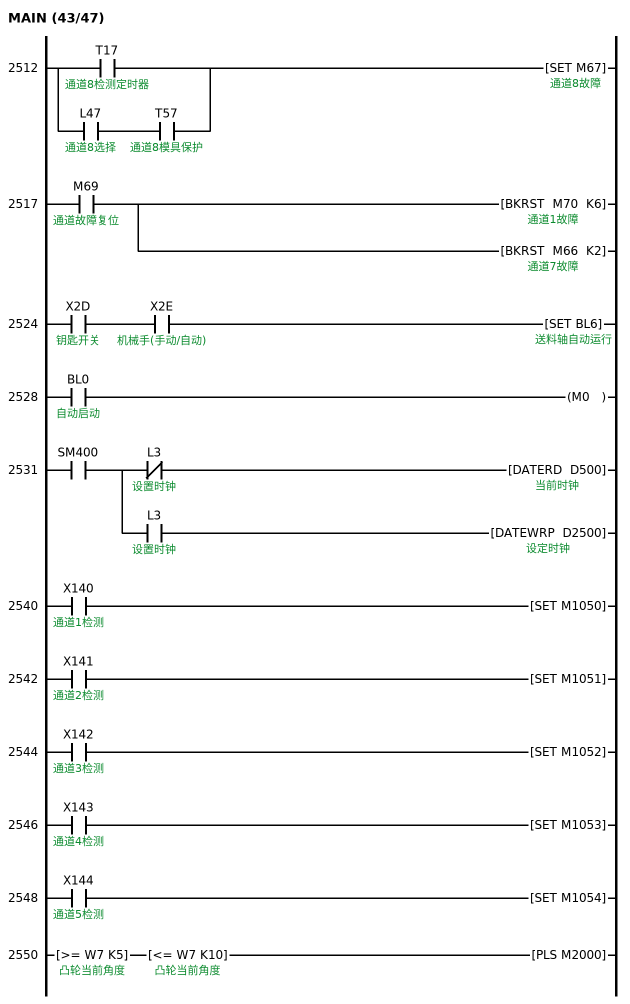
2512  LD      T17  ; 通道8检测定时器
      LD      L47  ; 通道8选择
      AND     T57  ; 通道8模具保护
      ORB
      SET     M67  ; 通道8故障
2517  LD      M69  ; 通道故障复位
      BKRST   M70 K6
      BKRST   M66 K2
2524  LD      X2D  ; 钥匙开关
      AND     X2E  ; 机械手(手动/自动)
      SET     BL6  ; 送料轴自动运行
2528  LD      BL0  ; 自动启动
      OUT     M0
2531  LD      SM400
      MPS
      ANI     L3  ; 设置时钟
      DATERD  D500  ; 当前时钟
      MPP
      AND     L3  ; 设置时钟
      DATEWRP D2500  ; 设定时钟
2540  LD      X140  ; 通道1检测
      SET     M1050
2542  LD      X141  ; 通道2检测
      SET     M1051
2544  LD      X142  ; 通道3检测
      SET     M1052
2546  LD      X143  ; 通道4检测
      SET     M1053
2548  LD      X144  ; 通道5检测
      SET     M1054
2550  LD>=    W7 K5  ; 凸轮当前角度
      AND<=   W7 K10  ; 凸轮当前角度
      PLS     M2000
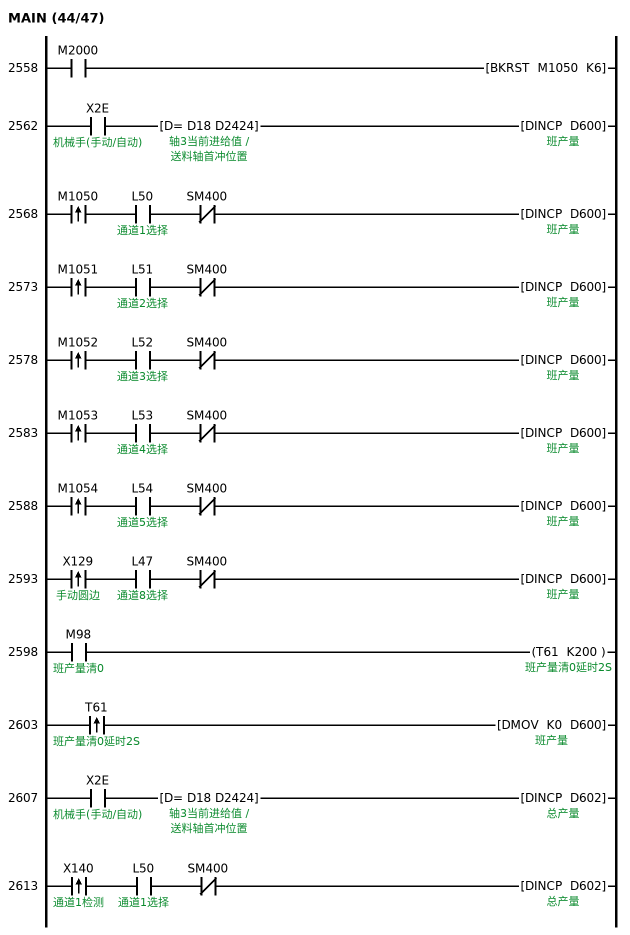
2558  LD      M2000
      BKRST   M1050 K6
2562  LD      X2E  ; 机械手(手动/自动)
      ANDD=   D18 D2424  ; 轴3当前进给值 / 送料轴首冲位置
      DINCP   D600  ; 班产量
2568  LDP     M1050
      AND     L50  ; 通道1选择
      ANI     SM400
      DINCP   D600
2573  LDP     M1051
      AND     L51  ; 通道2选择
      ANI     SM400
      DINCP   D600
2578  LDP     M1052
      AND     L52  ; 通道3选择
      ANI     SM400
      DINCP   D600
2583  LDP     M1053
      AND     L53  ; 通道4选择
      ANI     SM400
      DINCP   D600
2588  LDP     M1054
      AND     L54  ; 通道5选择
      ANI     SM400
      DINCP   D600
2593  LDP     X129  ; 手动圆边
      AND     L47  ; 通道8选择
      ANI     SM400
      DINCP   D600
2598  LD      M98  ; 班产量清0
      OUT     T61 K200  ; 班产量清0延时2S
2603  LDP     T61  ; 班产量清0延时2S
      DMOV    K0 D600
2607  LD      X2E  ; 机械手(手动/自动)
      ANDD=   D18 D2424  ; 轴3当前进给值 / 送料轴首冲位置
      DINCP   D602  ; 总产量
2613  LDP     X140  ; 通道1检测
      AND     L50  ; 通道1选择
      ANI     SM400
      DINCP   D602
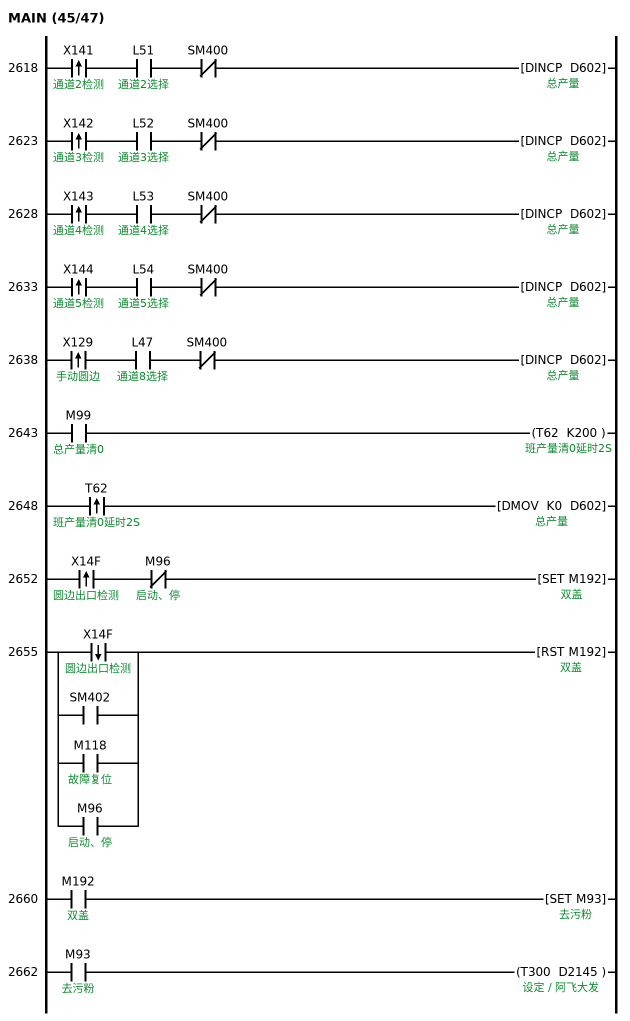
2618  LDP     X141  ; 通道2检测
      AND     L51  ; 通道2选择
      ANI     SM400
      DINCP   D602
2623  LDP     X142  ; 通道3检测
      AND     L52  ; 通道3选择
      ANI     SM400
      DINCP   D602
2628  LDP     X143  ; 通道4检测
      AND     L53  ; 通道4选择
      ANI     SM400
      DINCP   D602
2633  LDP     X144  ; 通道5检测
      AND     L54  ; 通道5选择
      ANI     SM400
      DINCP   D602
2638  LDP     X129  ; 手动圆边
      AND     L47  ; 通道8选择
      ANI     SM400
      DINCP   D602
2643  LD      M99  ; 总产量清0
      OUT     T62 K200  ; 班产量清0延时2S
2648  LDP     T62  ; 班产量清0延时2S
      DMOV    K0 D602
2652  LDP     X14F  ; 圆边出口检测
      ANI     M96  ; 启动、停
      SET     M192  ; 双盖
2655  LDF     X14F  ; 圆边出口检测
      OR      SM402
      OR      M118  ; 故障复位
      OR      M96  ; 启动、停
      RST     M192  ; 双盖
2660  LD      M192  ; 双盖
      SET     M93  ; 去污粉
2662  LD      M93  ; 去污粉
      OUTH    T300 D2145  ; 设定 / 阿飞大发
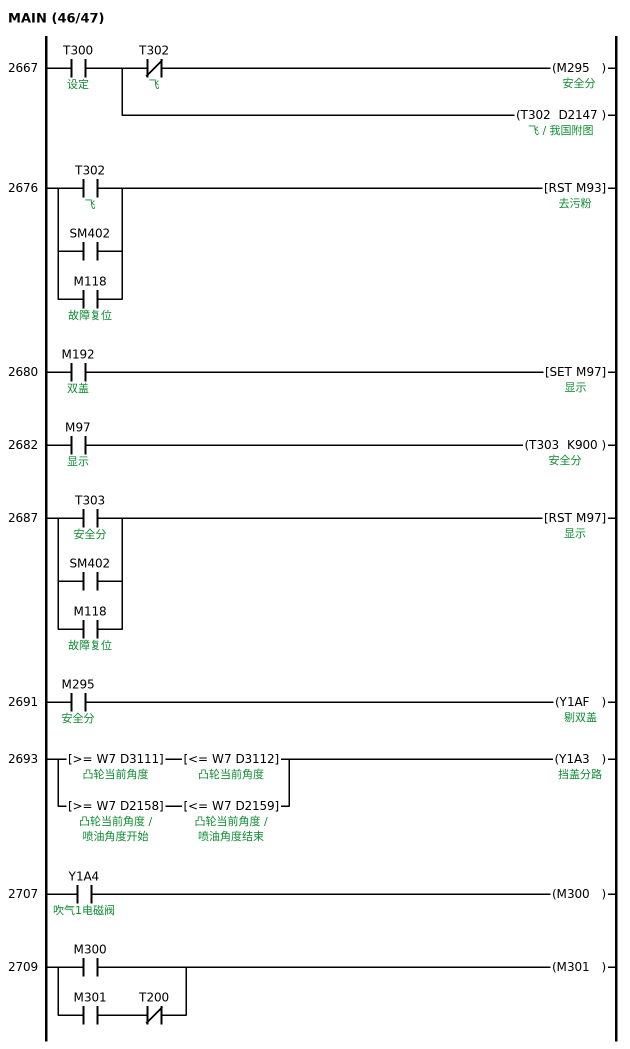
2667  LD      T300  ; 设定
      MPS
      ANI     T302  ; 飞
      OUT     M295  ; 安全分
      MPP
      OUTH    T302 D2147  ; 飞 / 我国附图
2676  LD      T302  ; 飞
      OR      SM402
      OR      M118  ; 故障复位
      RST     M93  ; 去污粉
2680  LD      M192  ; 双盖
      SET     M97  ; 显示
2682  LD      M97  ; 显示
      OUT     T303 K900  ; 安全分
2687  LD      T303  ; 安全分
      OR      SM402
      OR      M118  ; 故障复位
      RST     M97  ; 显示
2691  LD      M295  ; 安全分
      OUT     Y1AF  ; 剔双盖
2693  LD>=    W7 D3111  ; 凸轮当前角度
      AND<=   W7 D3112  ; 凸轮当前角度
      LD>=    W7 D2158  ; 凸轮当前角度 / 喷油角度开始
      AND<=   W7 D2159  ; 凸轮当前角度 / 喷油角度结束
      ORB
      OUT     Y1A3  ; 挡盖分路
2707  LD      Y1A4  ; 吹气1电磁阀
      OUT     M300
2709  LD      M300
      LD      M301
      ANI     T200
      ORB
      OUT     M301
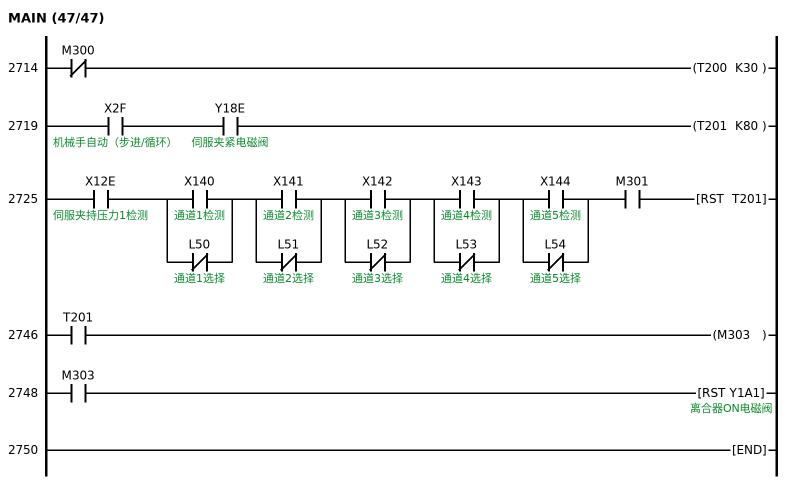
2714  LDI     M300
      OUT     T200 K30
2719  LD      X2F  ; 机械手自动（步进/循环）
      AND     Y18E  ; 伺服夹紧电磁阀
      OUT     T201 K80
2725  LD      X12E  ; 伺服夹持压力1检测
      LD      X140  ; 通道1检测
      ORI     L50  ; 通道1选择
      ANB
      LD      X141  ; 通道2检测
      ORI     L51  ; 通道2选择
      ANB
      LD      X142  ; 通道3检测
      ORI     L52  ; 通道3选择
      ANB
      LD      X143  ; 通道4检测
      ORI     L53  ; 通道4选择
      ANB
      LD      X144  ; 通道5检测
      ORI     L54  ; 通道5选择
      ANB
      AND     M301
      RST     T201
2746  LD      T201
      OUT     M303
2748  LD      M303
      RST     Y1A1  ; 离合器ON电磁阀
2750  END
END_PROGRAM

// device comments not shown above
M3  ; 允许手动开伺服
M7  ; 离合器ON/OFF指令（手动时）
M8  ; 离合器ON/OFF(自动启动)
M100  ; 强制启动分张机构
M112  ; tuy
M115  ; 送片延时
M190  ; 提前启动片料抬升
M250  ; 中文
M251  ; 英文
M412  ; 1s
M1001  ; 凸轮当前值<=离合器OFF角度
M1011  ; 首冲前位置
M6008  ; 模拟喷油信号
L0  ; 60度/90度  OFF方孔
L20  ; X轴奇数排移动方向
L21  ; X轴偶数排移动方向
L22  ; X轴寄到偶移动方向
L23  ; X轴偶到寄移动方向
L42  ; 顶料允许/禁止
L57  ; 主通风电机允许/禁止
X61  ; 绝地值编码器2
X62  ; 绝地值编码器3
X63  ; 绝地值编码器4
X64  ; 绝地值编码器5
X65  ; 绝地值编码器6
X66  ; 绝地值编码器7
X67  ; 绝地值编码器8
X68  ; 绝地值编码器9
X69  ; 绝地值编码器10
X103  ; 分张后吸上1到位
X104  ; 分张后吸上2到位
X105  ; 分张前吸上1到位
X106  ; 分张前吸上2到位
X107  ; 分张前吸上3到位
X108  ; 分张送料到位
X109  ; 分张送料复位
X10D  ; 分张后吸电磁阀下到位
X10F  ; 分张前吸电磁阀下到位
X120  ; 工作台落料到位
X122  ; 工作台右后定位
X123  ; 工作台测定位
X127  ; 抓手合拢压力检测
X128  ; 工作台抬升下到位
X12A  ; 工作台送料到前检测
X12C  ; 工作台左后定位
X14B  ; 排废料上限位
Y3F  ; 变频器复位
Y0E0  ; 变频正转启动
Y1032  ; 真空泵电机手动
Y1034  ; 主通风电机手动
Y103A  ; 圆边电机2手动
Y1181  ; 手动落料吸电磁阀
Y1182  ; 手动向后定位电磁阀
Y1183  ; 手动向侧定位电磁阀
Y11A3  ; 手动喷油
D36  ; X轴当前启动编号
D37  ; Y轴当前启动编号
D39  ; 轴1当前状态
D40  ; 轴2当前状态
D100  ; X轴0度定位长度D+间隔
D102  ; X轴0度定位长度（D+间隔）浮点数
D104  ; 定位角度转换浮点数
D106  ; 定位角度转换为弧度
D108  ; SIN60度
D110  ; COS60度
D112  ; Y轴定位长度浮点数
D114  ; X轴定位长度（差补）浮点数
D118  ; X轴定位长度差补（D+间隔）COS60
D120  ; D/2
D124  ; Ye
D126  ; 第一冲前定位长度Yo+Ye
D136  ; m-1排浮点数
D138  ; m排浮点数
D140  ; m排
D150  ; n-1列浮点数
D152  ; n列浮点数
D154  ; n列
D156  ; 冲片直径D浮点数
D158  ; m排浮点数
D160  ; n列浮点数
D162  ; 片材长度浮点数
D164  ; 片材宽度浮点数
D182  ; 冲片效率
D184  ; X轴0度定位长度负值-（D+间隔）
D188  ; X轴定位长度（差补）负值
D192  ; l-L
D194  ; l-L+l1
D206  ; 1路径定位X2
D208  ; 1路径定位X3
D210  ; 1路径定位X4
D212  ; 2路径定位X2
D214  ; 2路径定位X3
D216  ; 2路径定位X4
D218  ; 第三路径第2定位
D220  ; 第三路径第3定位
D222  ; 第三路径第4定位
D224  ; 第三路径第5定位
D226  ; 第三路径第6定位
D228  ; 第1，2路径最大行程
D240  ; 3路径首冲前定位位置
D244  ; 1路径定位X1
D246  ; 2路径定位X1
D248  ; 3路径定位X1
D262  ; 飞轮转速检测(脉冲数/1mim)
D2028  ; X轴奇数排移动次数
D2030  ; X轴偶数排移动次数
D2038  ; Yo第一冲模具长度参数
D2044  ; 片材宽度
D2046  ; 片材长度L
D2050  ; 冲几排开始向前送料
D2108  ; 剔废ON角度
D2110  ; 剔废OFF角度
D2138  ; X轴奇数排平移当前循环次数
D2140  ; X轴偶数排平移当前循环次数
D2142  ; 循环X轴定位位置
D2150  ; 当前循环次数
D2152  ; 循环Y轴定位位置
T5  ; 喷油时间
T6  ; 有料检测后延时1S(确保料稳定)
T7  ; 送片延时
T8  ; 后定位到延时100ms
T20  ; 吸料延时(确保料吸住)
T21  ; 后定位，测定位结束延时100ms
T22  ; 挡料缸落下和夹紧延时100ms
T24  ; 定位夹手到位，可以送料延时100ms
T30  ; 延时
T33  ; 夹紧延时
T43  ; 翻板ON延时100ms
T45  ; 首冲启动延迟摆动时间
T88  ; 双盖
T92  ; 工作台有料延时
